FUNCTION_BLOCK FB_DataChannelSenderFifo EXTENDS FB_DynamicFifo
VAR_INPUT
END_VAR
VAR_OUTPUT
END_VAR
VAR
	m_pDataChannel				: POINTER TO FB_DataChannelSendBase;
	m_pItem						: POINTER TO BYTE;
	m_bolEnable					: BOOL;
	m_intMaxFifoSize			: INT  	:= 10;
	
	bResult						: BOOL;
END_VAR

IF (m_uinItemCount > 0) AND NOT m_pDataChannel^.Busy THEN
	m_pItem := Pop();

	IF m_bolEnable THEN
		bResult := m_pDataChannel^.SendData(
						pData       := m_pItem,
						udiDataSize := m_pDataChannel^.DataSize);
	END_IF;
	
	IF m_bFreeDataPointer THEN
		__DELETE(m_pItem); 
	END_IF
END_IF

m_pDataChannel^();

PROPERTY PUBLIC DataChannel : POINTER TO FB_DataChannelSendBase
SET
m_pDataChannel := DataChannel;
END_SET
END_PROPERTY

PROPERTY PUBLIC Enable : BOOL
GET
Enable := m_bolEnable;
END_GET
SET
IF m_bolEnable AND NOT Enable THEN
	THIS^.ClearFifo();
END_IF

m_bolEnable := Enable;
END_SET
END_PROPERTY

PROPERTY PUBLIC MaxFifoSize : INT
GET
MaxFifoSize := m_intMaxFifoSize;
END_GET
SET
m_intMaxFifoSize := MaxFifoSize;
END_SET
END_PROPERTY

END_FUNCTION_BLOCK

(* stored: Version 1.1.0.1, ProductVersion 3.1.0.24
   POU FB_DataChannelSenderFifo: Id {7165605f-18c7-4e50-90e1-6b86acd60fdb}
   Property DataChannel: Id {6bb6fc5e-5fe4-4045-91d2-19a5787b0931}
   Set Set: Id {b268b1fd-b00e-422c-9c09-bb9fcdb55b14}
   Property Enable: Id {ac1ec63b-6014-4ada-8b4b-9a468375afbe}
   Get Get: Id {6ec7a47e-8020-4ad7-be76-1efbc6e7c75f}
   Set Set: Id {8447f007-3f1b-4e26-9ee9-899131542dda}
   Property MaxFifoSize: Id {f9b7a10f-2fa4-4593-b0fe-90a8b1176b52}
   Get Get: Id {a61726e9-fdf2-4fe1-aab5-65df90a17a58}
   Set Set: Id {fea3bb87-c11e-4073-b75e-30390707b124} *)
